// TwinCAT 3 PLC project L2SIVacuum
// Title: LCLS Vacuum
// Company: SLAC - LCLS
// Author: LCLS ECS-Platforms
// ProjectVersion: 0.0.0
// ProgramVersion: 3.1.4026.17
// libraries:
//   LCLS General, * (SLAC)
//   PMPS, * (SLAC - LCLS)
//   Tc2_DataExchange, * (Beckhoff Automation GmbH)
//   Tc2_EtherCAT, * (Beckhoff Automation GmbH)
//   Tc2_ModbusSrv, * (Beckhoff Automation GmbH)
//   Tc2_SerialCom, * (Beckhoff Automation GmbH)
//   Tc2_Standard, * (Beckhoff Automation GmbH)
//   Tc2_System, * (Beckhoff Automation GmbH)
//   Tc2_TcpIp, * (Beckhoff Automation GmbH)
//   Tc2_Utilities, * (Beckhoff Automation GmbH)
//   Tc3_EventLogger, * (Beckhoff Automation GmbH)
//   Tc3_JsonXml, * (Beckhoff Automation GmbH)
//   Tc3_Module, * (Beckhoff Automation GmbH)
//   TcUnit, * (www.tcunit.org)
// project tree:
//   DUTs/Gauges/ E_PressureState.TcDUT (not stored), Gauge_Type.TcDUT (not stored), ST_VG.TcDUT (not stored)
//   DUTs/LVDT/ ST_SerLVC4000.TcDUT (not stored)
//   DUTs/Oerlikon/ ST_TD20Status.TcDUT (not stored), ST_TD400Control.TcDUT (not stored), ST_TD400Status.TcDUT (not stored)
//   DUTs/Pfeiffer/ ST_PfeifferControl.TcDUT (not stored), ST_PfeifferStatus.TcDUT (not stored)
//   DUTs/Pumps/ E_PumpState.TcDUT (not stored), ST_AgilentPTM.TcDUT (not stored), ST_EbaraDryPump.TcDUT (not stored), ST_EbaraEVA.TcDUT (not stored), ST_EbaraPTM.TcDUT (not stored), ST_KashiyamaDryPump.TcDUT, ST_LeyboldPTM.TcDUT (not stored), ST_PfeifferPTM.TcDUT (not stored), ST_PIP.TcDUT (not stored), ST_PTM.TcDUT (not stored), ST_RoughPump.TcDUT (not stored)
//   DUTs/Valves/ E_ValvePositionState.TcDUT (not stored), E_VCN.TcDUT (not stored), E_2OO3_MODE.TcDUT (not stored), E_VGC.TcDUT (not stored), ST_ValveBase.TcDUT (not stored), ST_VFS.TcDUT (not stored), ST_VGC_2S.TcDUT (not stored), ST_VRC_NO.TcDUT (not stored), ST_VWC_NO.TcDUT (not stored), ST_VVC.TcDUT (not stored), ST_VCC_NO.TcDUT (not stored), ST_VCN.TcDUT (not stored), ST_VGC.TcDUT (not stored), ST_VRC.TcDUT (not stored)
//   DUTs/Valves/VAT590/EtherCAT Interface/ E_ControlMode.TcDUT (not stored), E_ControlModeSP.TcDUT (not stored), E_FatalErrors.TcDUT (not stored), ST_ExtendedWarnings.TcDUT (not stored), ST_GeneralControlSP.TcDUT (not stored), ST_GeneralStatus.TcDUT (not stored), ST_GeneralWarnings.TcDUT (not stored)
//   DUTs/Valves/VAT590/ E_VAT590_AccessMode.TcDUT (not stored), E_VAT590_PID_CTRL.TcDUT (not stored), E_VCN_VAT590.TcDUT (not stored), ST_CoEIndSub.TcDUT (not stored), ST_VAT590_COE.TcDUT (not stored), ST_VAT590_STATUS.TcDUT (not stored), ST_VCN_VAT590.TcDUT (not stored)
//   GVLs/ Constants.TcGVL (not stored), Global_Variables.TcGVL (not stored), GVL_MacroSensorsParameters.TcGVL (not stored), GVL_PfeifferParameters.TcGVL (not stored)
//   / PlcTask.TcTTO (not stored)
//   POUs/ADS/ FB_ADS.TcPOU (not stored), FB_ADS_WATCHDOG.TcPOU (not stored), FB_TBOOL_ADS.TcPOU (not stored)
//   POUs/Functions/Deprecated/Gauges/ FB_MKS317A.TcPOU (not stored), FB_MKS500_EP.TcPOU (not stored), FB_PressureState.TcPOU (not stored)
//   POUs/Functions/Deprecated/Valves/ FB_VCC.TcPOU (not stored), FB_VCC_NO.TcPOU (not stored), FB_VGC_AP.TcPOU (not stored), FB_VGC_EBD.TcPOU (not stored)
//   POUs/Functions/Gauges/ FB_901_ECAT.TcPOU (not stored), FB_9XX.TcPOU (not stored), FB_972.TcPOU (not stored), FB_IE514.TcPOU (not stored), FB_MX7M.TcPOU (not stored), FB_MKS355.TcPOU (not stored), FB_GaugeBase.TcPOU (not stored), FB_CVM201.TcPOU (not stored), FB_CCM501.TcPOU (not stored), FB_IMG401.TcPOU (not stored), FB_MKS909.TcPOU, FB_MKS909_RBK.TcPOU (not stored), FB_CMR362.TcPOU (not stored), FB_GCM.TcPOU (not stored), FB_ITR90.TcPOU (not stored), FB_MKS392.TcPOU (not stored), FB_MKS500.TcPOU (not stored), FB_MKS722.TcPOU (not stored), FB_MKS_937A.TcPOU (not stored), FB_MKS317.TcPOU (not stored), FB_MKS275.TcPOU (not stored), FB_MKS_937B.TcPOU (not stored), FB_MKS422.TcPOU (not stored)
//   POUs/Functions/Gauges/Interfaces/ FB_GaugeModbus.TcPOU (not stored), FB_Gauge_Interface.TcPOU, FB_TGCC_ADS.TcPOU (not stored), FB_TGPI_ADS.TcPOU (not stored), FB_GaugeSelection.TcPOU
//   POUs/Functions/Pumps/ FB_EbaraDryPump.TcPOU (not stored), FB_EbaraEVA.TcPOU (not stored), FB_KashiyamaPump.TcPOU, FB_KashiyamaPump_G.TcPOU, FB_PIP_Gamma.TcPOU (not stored), FB_PIP_SIP.TcPOU (not stored), FB_PTM_Agilent.TcPOU (not stored), FB_PTM_Ebara_011M.TcPOU (not stored), FB_PTM_Ebara_010M.TcPOU (not stored), FB_PTM_MagDriveDigital.TcPOU (not stored), FB_PTM_Pfeiffer.TcPOU (not stored), FB_PTM_TurboDrive.TcPOU (not stored), FB_PTM_TwisTorr.TcPOU (not stored), FB_Pump.TcPOU (not stored), FB_ScrollPump.TcPOU (not stored)
//   POUs/Functions/Pumps/functions/ FB_TurboExtLogic.TcPOU (not stored), F_TurboExtILK_NO.TcPOU (not stored), F_TurboExtILKLogic.TcPOU (not stored), F_TurboExtILKLogic_2.TcPOU (not stored), F_TurboExtILK_NO_1.TcPOU (not stored)
//   POUs/Functions/Pumps/Interfaces/ FB_PIP_Interface_In.TcPOU (not stored), FB_PIP_Interface_Out.TcPOU (not stored), FB_TPIP_ADS.TcPOU (not stored)
//   POUs/Functions/Valves/ FB_Kashiyama_VRC.TcPOU (not stored), FB_MKS248.TcPOU (not stored), FB_TurbVentvalve_NO.TcPOU (not stored), FB_Valve.TcPOU (not stored), FB_VCN_VAT590.TcPOU (not stored), FB_VFS.TcPOU (not stored), FB_VFS_2OO3.TcPOU (not stored), FB_VGC_2S.TcPOU (not stored), FB_VRC_DA.TcPOU (not stored), FB_VRC_EBD.TcPOU (not stored), FB_VRC_NC_ClsLS.TcPOU (not stored), FB_VRC_NO.TcPOU (not stored), FB_VRC_NO_FFO.TcPOU (not stored), FB_VVC.TcPOU (not stored), FB_VCN.TcPOU (not stored), FB_VGC.TcPOU (not stored), FB_VRC.TcPOU (not stored), FB_VRC_OK_CLS.TcPOU (not stored)
//   POUs/Functions/Valves/functions/ F_RoughPumpInlet_ILK.TcPOU (not stored), F_TurboGateValve_ILK.TcPOU (not stored), F_TurboGateValve_ILK_1.TcPOU (not stored), F_TurboGateValve_Protection_ILK.TcPOU (not stored), F_TURBO_VRC_ILK.TcPOU (not stored), F_VALVE_REL_ILK.TcPOU (not stored), F_VRC_DIODE_ILK_OK.TcPOU (not stored), F_VRC_DIODE_ILK.TcPOU (not stored)
//   POUs/Functions/Valves/Interfaces/ FB_TVGC_2S_ADS.TcPOU (not stored), FB_VFS_2OO3Interface.TcPOU (not stored), FB_VFS_Interface.TcPOU (not stored), FB_TVGC_ADS.TcPOU (not stored), FB_Valve_Interface.TcPOU (not stored), ITF_Valve.TcIO (not stored)
//   POUs/Serial drivers/LVDT/MacroSensors/ FB_LVC4000Com.TcPOU (not stored), FB_LVC4000SerialDriver.TcPOU (not stored), FB_LVC4000Transaction.TcPOU (not stored)
//   POUs/Serial drivers/Pumps/Oerlikon TD20/ FB_OERLIKON_TD20_COM.TcPOU (not stored), FB_OERLIKON_TO_PTM.TcPOU (not stored), FB_TD20SerialDriver.TcPOU (not stored), FB_TD20Transaction.TcPOU (not stored), F_CalcTD20Checksum.TcPOU (not stored)
//   POUs/Serial drivers/Pumps/Oerlikon TD400/ FB_OERLIKON_TD400_COM.TcPOU (not stored), FB_OERLIKON_TD400_TO_PTM.TcPOU (not stored), FB_TD400SerialDriver.TcPOU (not stored), FB_TD400Transaction.TcPOU (not stored), F_CalcTD400Checksum.TcPOU (not stored)
//   POUs/Serial drivers/Pumps/Pfeiffer/ FB_PfeifferSerialDriver.TcPOU (not stored), FB_PfeifferTransaction.TcPOU (not stored), FB_PFEIFFER_COM.TcPOU (not stored), FB_PFEIFFER_TO_PTM.TcPOU (not stored), F_CalcPfeifferCheckSum.TcPOU (not stored)
//   UnitTests/Functions/ V_TO_INT.TcPOU (not stored)
//   UnitTests/Gauges/ FB_GCC_Test.TcPOU (not stored), FB_GHC_Test.TcPOU (not stored), FB_GPI_Test.TcPOU (not stored)
//   UnitTests/ PRG_Test.TcPOU (not stored)
//   UnitTests/Pumps/ FB_PIP_Test.TcPOU (not stored), FB_PTM_Test.TcPOU (not stored)
//   UnitTests/Valves/ FB_VGC_Test.TcPOU (not stored), FB_VRC_Test.TcPOU (not stored)
//   Version/ Global_Version.TcGVL (not stored)
// real-time tasks:
//   TASK TestTask: cycle T#10ms, priority 16, ADS port 350
// variable links:
//   L2SIVacuum/L2SIVacuum Instance <-> L2SIVacuum/L2SIVacuum Instance
//     PlcTask Inputs/PRG_Test.fb_GCC_Test.fb_MKS422.i_iPRESS_R <-> PlcTask Outputs/PRG_Test.fb_GCC_Test.i_iPRESS_R
//     PlcTask Inputs/PRG_Test.fb_GPI_Test.fb_MKS275.i_iPRESS_R <-> PlcTask Outputs/PRG_Test.fb_GPI_Test.i_iPRESS_R
//     PlcTask Inputs/PRG_Test.fb_GPI_Test.fb_MKS317.i_iPRESS_R <-> PlcTask Outputs/PRG_Test.fb_GPI_Test.i_iPRESS_R
//     PlcTask Inputs/PRG_Test.fb_PTM_Test.fb_PTM_Ebara_010M.i_iCurrentMon <-> PlcTask Outputs/PRG_Test.fb_PTM_Test.i_iCurrentMon
//     PlcTask Inputs/PRG_Test.fb_PTM_Test.fb_PTM_Ebara_010M.i_iRawSpeed <-> PlcTask Outputs/PRG_Test.fb_PTM_Test.i_iRawSpeed
//     PlcTask Inputs/PRG_Test.fb_PTM_Test.fb_PTM_Ebara_010M.i_iTempMon <-> PlcTask Outputs/PRG_Test.fb_PTM_Test.i_iTempMon
//     PlcTask Inputs/PRG_Test.fb_PTM_Test.q_iSpeedSet <-> PlcTask Outputs/PRG_Test.fb_PTM_Test.i_diCurSpd

// ---- DUTs/Pumps/ST_KashiyamaDryPump.TcDUT
TYPE ST_KashiyamaDryPump EXTENDS ST_RoughPump:
STRUCT

(* Output *)
    //q_xRunDO 	:	BOOL; in Rough PUMP
    {attribute 'pytmc' := '
    pv: RESET_DO;
    field: ZNAM FALSE;
    field: ONAM TRUE;
    io: i
    '}
    q_xResetDo	: 	BOOL;
    {attribute 'pytmc' := '
    pv: LSPD_DO;
    field: ZNAM FALSE;
    field: ONAM TRUE;
    io: i
    '}
    q_xLspdDo	: 	BOOL;
    {attribute 'pytmc' := '
    pv: REM_DO;
    field: ZNAM FALSE;
    field: ONAM TRUE;
    io: i
    '}
    q_xRemoteDo	: 	BOOL;

(* Input *)
{attribute 'pytmc' := '
    pv: REMOTE;
    field: ZNAM FALSE;
    field: ONAM TRUE;
    io: i
    '}
    i_xRemote	:	BOOL;

    {attribute 'pytmc' := '
    pv: ALARM_OK;
    field: ZNAM FALSE;
    field: ONAM TRUE;
    io: i
    '}
    i_xAlarmOK	:	BOOL;
    {attribute 'pytmc' := '
    pv: WARN_OK;
    field: ZNAM FALSE;
    field: ONAM TRUE;
    io: i
    '}
    i_xWarningOK	:	BOOL;
    {attribute 'pytmc' := '
    pv: RUN_DI;
    field: ZNAM FALSE;
    field: ONAM TRUE;
    io: i
    '}
    i_xIsRun		:	BOOL;

(* Logic status *)

    xLspd_IlkENA:   BOOL;

(* EPICS *)
    //xRunSW		:	BOOL; in Rough PUMP
    {attribute 'pytmc' := '
    pv: RESET_SW;
    field: ZNAM FALSE;
    field: ONAM TRUE;
    io: io
    '}
    xResetSW	:	BOOL; //For resetting faults
    {attribute 'pytmc' := '
    pv: LSPD_SW;
    field: ZNAM FALSE;
    field: ONAM TRUE;
    io: io
    '}
    xLspdSW     :   BOOL;
    {attribute 'pytmc' := '
    pv: REMOTE_SW;
    field: ZNAM FALSE;
    field: ONAM TRUE;
    io: io
    '}
    xRemoteSW     :   BOOL;
    LowSP  :   REAL := 0.02; //Torr
    HighSP :   REAL; //Torr
    RdyTmr : REAL;
END_STRUCT
END_TYPE

// ---- POUs/Functions/Gauges/FB_MKS909.TcPOU
(* Standard MKS 909 hot cathode *)
(* works for 972 and 925 *)

FUNCTION_BLOCK FB_MKS909 EXTENDS FB_GaugeBase

VAR_INPUT
    PG	: ST_VG;
END_VAR
VAR_OUTPUT
    {attribute 'pytmc' := '
    pv:
    '}
    IG	: ST_VG;
END_VAR
VAR_IN_OUT

END_VAR
VAR
    rV : REAL;
    rMaxPressure	:	REAL := 5E-2; //Torr
    rMinPressure	:	REAL := 1E-10; //Torr
    timer:TON;
    (*Default set point 50 mT*)
    rDefaultVAC_SP: REAL := 9E-3; // as per manual
    iTermBits: UINT := 30518 ; // The terminal's maximum value in bits default el3174 as per vacuum architecture
    (*IO*)
    i_iPRESS_R AT%I* :INT; // input Pressure // Link to analog Input
    q_xHV_DIS AT %Q* : BOOL := True; // Active Low
    i_xHV_ON AT %I*	: BOOL; //  True when High Voltage is on  // 'TcLinkTo' (EL1084) ^Input

END_VAR

(* Standard MKS 9XX series conversion *)
(* works for 972 and 925 *)

//Default setpoint 50 mT
IF PG.rVAC_SP = 0 THEN
    PG.rVAC_SP := rDefaultVAC_SP;
END_IF
// check no div by zero
If (iTermBits=0) THEN iTermBits := 30518;END_IF
rV := 10*INT_TO_REAL(IG.i_iPRESS_R)/iTermBits;

(* Pressure OK check *)
// Gauge state
// Is the gauge plugged in, and within a reasonable range?
IF  (rV >= 0.1 and rV <=8.7) AND IG.i_xHV_ON THEN // as per manual
    IG.rPRESS := LREAL_TO_REAL(EXPT(10, rV-10));
    IG.eState := Valid;
    IG.xPRESS_OK := TRUE; //Backwards compatibility
ELSIF rV > 8.7 AND rV < 10 AND IG.i_xHV_ON THEN
    IG.rPRESS :=rMaxPressure;
    IG.xPRESS_OK := FALSE;
    IG.eState := Off;
ELSE
    IG.xPRESS_OK := FALSE;
    IG.eState := GaugeDisconnected;
END_IF


IF (PG.rPRESS <= IG.rPRO_SP)  AND (PG.xPRESS_OK) THEN
         IG.q_xHV_DIS := IG.xHV_SW;
         IG.xILKOk := TRUE;
    ELSIF NOT IG.q_xHV_DIS AND timer.Q THEN
        IF IG.rPRESS > (IG.rPRO_SP + IG.rHYS_PR) OR PG.rPRESS > (IG.rPRO_SP + IG.rHYS_PR) THEN
        IG.q_xHV_DIS := FALSE;
        IG.xHV_SW := FALSE;
        END_IF
    ELSE
        IG.q_xHV_DIS := FALSE;
        IG.xHV_SW := FALSE;
        IG.xILKOk := FALSE;
     END_IF


timer(IN:= NOT IG.q_xHV_DIS, PT:= T#2s);

(* Setpoint evaluation *)
IG.xAT_VAC := IG.xPRESS_OK AND (IG.rPRESS < IG.rVAC_SP);

(*Soft IO Mapping*)
ACT_IO();
(*Load or save the persistent variables*)
ACT_Persistent();

(*Logger*)
THIS^.ACT_Logger();

(*Load or save the persistent variables*)
ACT_Persistent();

ACTION ACT_IO:
(*soft link inputs*)
IG.i_iPRESS_R:=	i_iPRESS_R;

(*soft link outputs*)
q_xHV_DIS := IG.q_xHV_DIS;
END_ACTION

ACTION ACT_Logger:
// ILK logger
IF NOT IG.xILKOk AND NOT IG.q_xHV_DIS THEN
         fbLogger(sMsg:='Lost external interlock while gauge was on.', eSevr:=TcEventSeverity.Critical);
END_IF


// Log Action
tAction(CLK:=  IG.q_xHV_DIS);
IF tAction.Q THEN fbLogger(sMsg:='Ion gauge commanded to switch on', eSevr:=TcEventSeverity.Info); END_IF



//STATE Logger
IF ePrevState <> IG.eState THEN
      CASE IG.eState OF
        ValidHi:
        ValidLo:
        Valid:
            fbLogger(sMsg:='Gauge pressure valid.', eSevr:=TcEventSeverity.Info);
          GaugeDisconnected:
            fbLogger(sMsg:='Gauge Disconnected.', eSevr:=TcEventSeverity.Critical);
        PressInvalid:
            fbLogger(sMsg:='Gauge pressure invalid.', eSevr:=TcEventSeverity.Warning);
        OoR:
            fbLogger(sMsg:='Gauge pressure out of range.', eSevr:=TcEventSeverity.Warning);
        Starting:
            fbLogger(sMsg:='Gauge starting.', eSevr:=TcEventSeverity.Info);
      END_CASE
      ePrevState := IG.eState;
END_IF
END_ACTION

ACTION ACT_Persistent:
(*On first PLC pass, load the persistent value into the structrue variable*)
IF (SUPER^.bRestorePersistentData) THEN
    SUPER^.bRestorePersistentData	:= FALSE;
    IF ( rVAC_SP <> 0) THEN
        IG.rVAC_SP := rVAC_SP;
    END_IF;
    IF ( rPRO_SP <> 0) THEN
        IG.rPRO_SP := rPRO_SP;
    END_IF;
    IF ( rHYS_PR <> 0) THEN
        IG.rHYS_PR := rHYS_PR;
    END_IF;
END_IF
(*Check if a new value has been written in the structure variable copy it to the persistent variable*)
IF NOT (IG.rVAC_SP = rVAC_SP)  THEN
    rVAC_SP := IG.rVAC_SP;
END_IF;

IF NOT (IG.rPRO_SP = rPRO_SP) THEN
    rPRO_SP:= IG.rPRO_SP;
END_IF;

IF NOT (IG.rHYS_PR = rHYS_PR) THEN
    rHYS_PR:= IG.rHYS_PR;
END_IF;
END_ACTION

METHOD M_AutoOn : BOOL
VAR_INPUT
END_VAR
this^.IG.q_xHV_DIS:= FALSE;
END_METHOD

METHOD M_SetBits : BOOL
VAR_INPUT
    TermBits : UINT; // The terminal's maximum value in bits
END_VAR
This^.iTermBits := TermBits;
END_METHOD

END_FUNCTION_BLOCK

// ---- POUs/Functions/Gauges/Interfaces/FB_Gauge_Interface.TcPOU
(* This function block is created for interface devices between different PLC*)
(* Not all the Variables in the original structure is required, just few signals *)
(* They have to be linked to the custom created variables on the EL6692/5 primary side*)
FUNCTION_BLOCK FB_Gauge_Interface
VAR_INPUT
END_VAR
VAR_OUTPUT
    {attribute 'pytmc' := 'pv:'}
    VG : ST_VG;
END_VAR
VAR
    i_rPRESS AT%I*: REAL;
    i_xAT_VAC AT%I*: BOOL;
    i_xPRESS_OK AT%I*: BOOL;
    i_sPath AT%I* : STRING;

END_VAR

(* This function block is created for interface devices between different PLC*)
(* Not all the Variables in the original structure is required, just few signals *)
(* They have to be linked to the custom created variables on the EL6692/5 primary side*)

VG.rPRESS := i_rPRESS;
VG.xAT_VAC := i_xAT_VAC;
VG.xPRESS_OK := i_xPRESS_OK;
VG.sPath := i_sPath;

END_FUNCTION_BLOCK

// ---- POUs/Functions/Gauges/Interfaces/FB_GaugeSelection.TcPOU
FUNCTION_BLOCK FB_GaugeSelection EXTENDS FB_GaugeBase
VAR_INPUT
    st_defaultGauge : ST_VG;
    st_secondGauge : ST_VG;
END_VAR
VAR_OUTPUT
    IG : ST_VG;
END_VAR
VAR
END_VAR

IF NOT st_defaultGauge.xPRESS_OK AND st_secondGauge.xPRESS_OK THEN
    IG := st_secondGauge;
ELSE
    IG := st_defaultGauge;
END_IF

END_FUNCTION_BLOCK

// ---- POUs/Functions/Pumps/FB_KashiyamaPump.TcPOU
(* This function block does basic controls FOR the Kashiyama pump. Turns off pump
in the event of errors/ warnings. Provides interlocking interface.*)
FUNCTION_BLOCK FB_KashiyamaPump
VAR_IN_OUT

END_VAR
VAR_INPUT

END_VAR
VAR_OUTPUT
    {attribute 'pytmc' := 'pv:'}
    q_stPump : ST_KashiyamaDryPump;
END_VAR
VAR
    TONtmr : TON;
    resetTmr : TON;

    (* Output *)
    q_xRunDO 	AT%Q*:	BOOL;
    q_xResetDo	AT%Q*: 	BOOL;
    q_xLspdDo	AT%Q*: 	BOOL;

(* Input *)
    i_xRemote	AT%I*:	BOOL;
    i_xAlarm	AT%I*:	BOOL;
    i_xWarning	AT%I*:	BOOL;
    i_xIsRun	AT%I*:	BOOL;
END_VAR


//Kashiyama Dry pump outputs at high level indicate no warning, no alarm and remotely
q_stPump.xIlkOK := q_stPump.i_xRemote AND q_stPump.i_xWarningOK AND q_stPump.i_xAlarmOK;

IF q_stPump.xIlkOK THEN
    q_stPump.q_xRunDO := q_stPump.pv_xRunSW;
    ELSE
        q_stPump.PV_xRunSW := FALSE;
        q_stPump.q_xRunDO := FALSE;
END_IF

q_stPump.xLspd_IlkENA := q_stPump.q_xRunDO;

IF q_stPump.xLspd_IlkENA THEN
    q_stPump.q_xLspdDo := q_stPump.xLspdSW;
    ELSE
        q_stPump.xLspdSW := FALSE;
        q_stPump.q_xLspdDo := FALSE;
END_IF

//resetTmr (In := iq_stPump.xResetSW, PT := T#2S);
//IF resetTmr.Q THEN
//	iq_stPump.xResetSW := FALSE;
//END_IF

q_stPump.q_xResetDo := NOT q_stPump.i_xIsRun AND q_stPump.xResetSW;

//countdown Timer
TONtmr (IN := q_stPump.i_xIsRun, PT := T#20S);
q_stPump.RdyTmr := TO_REAL(TONtmr.PT) - TO_REAL(TONtmr.ET);

(*State evaluation*)
IF NOT q_stPump.i_xAlarmOK THEN
    q_stPump.eState := pumpFAULT;
ELSIF NOT q_stPump.q_xRunDo AND q_stPump.i_xAlarmOK THEN
        q_stPump.eState := pumpSTOPPED;
ELSIF q_stPump.q_xRunDo AND NOT q_stPump.i_xIsRun THEN
        q_stPump.eState := pumpSTARTING;
ELSIF q_stPump.i_xIsRun THEN
        q_stPump.eState := pumpRUNNING;
ELSE
    q_stPump.eState := pumpFAULT;
END_IF

//Mapping
ACT_IO();

ACTION ACT_IO:
(* Output *)
    q_xRunDO 	:= q_stPump.q_xRunDO;
    q_xResetDo := q_stPump.q_xResetDo;;
    q_xLspdDo := q_stPump.q_xLspdDo;;

(* Input *)
    q_stPump.i_xRemote := i_xRemote;
    q_stPump.i_xAlarmOK :=	i_xAlarm;
    q_stPump.i_xWarningOK :=	i_xWarning;
    q_stPump.i_xIsRun :=	i_xIsRun;
END_ACTION

METHOD PUBLIC M_Run : BOOL
VAR_INPUT
    run:bool; // set to true to run, false to stop;
END_VAR

this^.q_stPump.pv_xRunSW := run;
END_METHOD

END_FUNCTION_BLOCK

// ---- POUs/Functions/Pumps/FB_KashiyamaPump_G.TcPOU
(* This function block does basic controls FOR the Kashiyama pump. Turns off pump
in the event of errors/ warnings. Provides interlocking interface.*)
FUNCTION_BLOCK FB_KashiyamaPump_G
VAR_IN_OUT

END_VAR
VAR_INPUT

END_VAR
VAR_OUTPUT
    {attribute 'pytmc' := 'pv:'}
    q_stPump : ST_KashiyamaDryPump;
END_VAR
VAR
    TONtmr : TON;
    resetTmr : TON;

    (* Output *)
    q_xRunDO 	AT%Q*:	BOOL;
    q_xResetDo	AT%Q*: 	BOOL;
    q_xLspdDo	AT%Q*: 	BOOL;
    q_xRemote 	AT%Q*:  BOOL;

(* Input *)
    i_xAlarm	AT%I*:	BOOL;
    i_xIsRun	AT%I*:	BOOL;
END_VAR


//Only run when commanded to be in remote and there is no alarm (this is a normally open alarm 0 = OK)
q_stPump.xIlkOK := q_stPump.q_xRemoteDO AND NOT q_stPump.i_xAlarmOK;

IF q_stPump.xIlkOK THEN
    q_stPump.q_xRunDO := q_stPump.pv_xRunSW;
    ELSE
        q_stPump.PV_xRunSW := FALSE;
        q_stPump.q_xRunDO := FALSE;
END_IF

q_stPump.xLspd_IlkENA := q_stPump.xIlkOK;

IF q_stPump.xLspd_IlkENA THEN
    q_stPump.q_xLspdDo := q_stPump.xLspdSW;
    ELSE
        q_stPump.xLspdSW := FALSE;
        q_stPump.q_xLspdDo := FALSE;
END_IF

//resetTmr (In := iq_stPump.xResetSW, PT := T#2S);
//IF resetTmr.Q THEN
//	iq_stPump.xResetSW := FALSE;
//END_IF

q_stPump.q_xResetDo := NOT q_stPump.i_xIsRun AND q_stPump.xResetSW;

//countdown Timer
TONtmr (IN := q_stPump.i_xIsRun, PT := T#20S);
q_stPump.RdyTmr := TO_REAL(TONtmr.PT) - TO_REAL(TONtmr.ET);

(*State evaluation*)
IF q_stPump.i_xAlarmOK THEN  // reminder this is normally closed (0 = no alarm | 1 = alarm)
    q_stPump.eState := pumpFAULT;
ELSIF NOT q_stPump.q_xRunDo AND NOT q_stPump.i_xAlarmOK THEN
        q_stPump.eState := pumpSTOPPED;
ELSIF q_stPump.q_xRunDo AND NOT q_stPump.i_xIsRun THEN
        q_stPump.eState := pumpSTARTING;
ELSIF q_stPump.i_xIsRun THEN
        q_stPump.eState := pumpRUNNING;
ELSE
    q_stPump.eState := pumpFAULT;
END_IF

//Mapping
M_IO();

METHOD M_Alarm : BOOL
VAR_INPUT
END_VAR
M_alarm := THIS^.q_stPump.i_xAlarmOK;   // 0 = no alarm | 1 = alarm
END_METHOD

METHOD M_IO : BOOL
VAR_INPUT
END_VAR
(* Output *)
    q_xRunDO 	:= THIS^.q_stPump.q_xRunDO;
    q_xResetDo := THIS^.q_stPump.q_xResetDo;
    q_xLspdDo := THIS^.q_stPump.q_xLspdDo;
    q_xRemote := THIS^.q_stPump.q_xRemoteDo;
(* Input *)
    THIS^.q_stPump.i_xAlarmOK :=	THIS^.i_xAlarm;
    THIS^.q_stPump.i_xIsRun :=	THIS^.i_xIsRun;
END_METHOD

METHOD M_IsRun : BOOL
VAR_INPUT
END_VAR
M_IsRun := THIS^.q_stPump.i_xIsRun;
END_METHOD

METHOD M_Lspd : BOOL
VAR_INPUT
    lowspeed : BOOL;  // Set low speed setting
END_VAR
THIS^.q_stPump.xLspdSW := lowspeed;
END_METHOD

METHOD M_Remote : BOOL
VAR_INPUT
    remote : BOOL; // Remote command
END_VAR
this^.q_stPump.xRemoteSW := remote;
END_METHOD

METHOD M_Reset : BOOL
VAR_INPUT
    reset : BOOL; // Set true to clear faults
END_VAR
this^.q_stPump.xResetSW := reset;
END_METHOD

METHOD PUBLIC M_Run : BOOL
VAR_INPUT
    run:bool; // set to true to run, false to stop;
END_VAR

this^.q_stPump.pv_xRunSW := run;
END_METHOD

END_FUNCTION_BLOCK
